Universal Robots PolyScope program: husarion_ext_control.urp

Program husarion_ext_control (installation=default directory=/programs createdIn=5.12.4.1101661 lastSavedIn=5.12.4.1101661 robotSerialNumber=20225590083)
Calibrated DH parameters: a=[-0.000014, -0.417005, -0.391941, -0.000072, 0.00008, 0]; d=[0.162637, -32.66166, 38.62048, -5.82524, 0.099855, 0.09965]; alpha=[1.570979, 0.002538, 0.003612, 1.570044, -1.570505, 0]; deltaTheta=[0, -0.196227, 6.53428, -0.054866, 0.000003, 0]
Robot Program (runOnlyOnce=false)
  URCap External Control (External Control, FZI Research Center for Information Technology)
Thread Thread_1 (runOnlyOnce=false)
  Wait Sleep waitTime=0.2
  Set ExpressionOutput pin=analog_out[1]; expression=get_rg_Width()/101.5
Thread Thread_2 (runOnlyOnce=false)
  Wait Condition expression=digital_out[0]≟ True
  Script: rg_grip((get_standard_analog_out(0)-0.0035)*6060, 40, tool_index = 0, blocking = True, depth_comp = False, popupmsg = True)
  Set DigitalOutput pin=digital_out[0]; digitalValue=0
